FUNCTION_BLOCK FB_RGBLED IMPLEMENTS ITF_SubSystem
VAR_INPUT
	eColor : LEDColor;
END_VAR
VAR
	//Local
	nRedLED : INT;
	nGreenLED : INT;
	nBlueLED : INT;
	
	aErrorTimer : ARRAY [0..5] OF TON;
	
	//ErrorBits
	bRedTemperatureTooHigh : BIT;
	bRedNoSupplyVoltage : BIT;
	bGreenTemperatureTooHigh : BIT;
	bGreenNoSupplyVoltage : BIT;
	bBlueTemperatureTooHigh : BIT;
	bBlueNoSupplyVoltage : BIT;	
END_VAR
VAR CONSTANT
	nMax : INT := 32767;		//Maximum Intensity (100%)
	nMin : INT := 0;			//Off (0%)
END_VAR

CASE eColor OF
	LEDColor.Off:
		nRedLED := nMin;
		nGreenLED := nMin;
		nBlueLED := nMin;
	LEDColor.Red:
		nRedLED := nMax;
		nGreenLED := nMin;
		nBlueLED := nMin;
	LEDColor.Green:
		nRedLED := nMin;
		nGreenLED := nMax;
		nBlueLED := nMin;
	LEDColor.Blue:
		nRedLED := nMin;
		nGreenLED := nMin;
		nBlueLED := nMax;
END_CASE



doSetClampValues();
doGetClampValues();

METHOD PRIVATE doGetClampValues
VAR_INPUT
END_VAR
bRedTemperatureTooHigh := RGBLED.bRedWarning;
bRedNoSupplyVoltage := RGBLED.bRedError;
bGreenTemperatureTooHigh := RGBLED.bGreenWarning;
bGreenNoSupplyVoltage := RGBLED.bGreenError;
bBlueTemperatureTooHigh := RGBLED.bBlueWarning;
bBlueNoSupplyVoltage := RGBLED.bBlueError;
END_METHOD

METHOD PRIVATE doSetClampValues
RGBLED.nRed := nRedLED;
RGBLED.nGreen := nGreenLED;
RGBLED.nBlue := nBlueLED;
END_METHOD

PROPERTY eCondition : SubLevelCondition
GET
IF nErrorID <> 0 THEN
	eCondition := SubLevelCondition.ERROR;
ELSE
	eCondition := SubLevelCondition.RUN;
END_IF
END_GET
END_PROPERTY

PROPERTY nErrorID : UDINT
GET
nErrorID.0 := aErrorTimer[0].Q;
nErrorID.1 := aErrorTimer[1].Q;
nErrorID.2 := aErrorTimer[2].Q;
nErrorID.3 := aErrorTimer[3].Q;
nErrorID.4 := aErrorTimer[4].Q;
nErrorID.5 := aErrorTimer[5].Q;

aErrorTimer[0](IN:=bRedTemperatureTooHigh, PT:=T#5S);
aErrorTimer[1](IN:=bRedNoSupplyVoltage, PT:=T#5S);
aErrorTimer[2](IN:=bGreenTemperatureTooHigh, PT:=T#5S);
aErrorTimer[3](IN:=bGreenNoSupplyVoltage, PT:=T#5S);
aErrorTimer[4](IN:=bBlueTemperatureTooHigh, PT:=T#5S);
aErrorTimer[5](IN:=bBlueNoSupplyVoltage, PT:=T#5S);
END_GET
END_PROPERTY

END_FUNCTION_BLOCK

(* stored: Version 1.1.0.1, ProductVersion 3.1.4024.12
   POU FB_RGBLED: Id {469ae6ce-499d-4fa3-8525-1529c7798012}, SpecialFunc None
   Method doGetClampValues: Id {52eec7f2-2131-4ede-95da-3597bc5e0c67}
   Method doSetClampValues: Id {dbe16808-2cac-4096-8234-89397ca2e1ed}
   Property eCondition: Id {07f8f374-c150-465f-b84c-fb20f0d2bc35}
   Get Get: Id {441c6c85-d8e3-4421-86d4-8b0d5eba7d41}
   Property nErrorID: Id {45849282-d051-426c-bf8e-7a781e21e522}
   Get Get: Id {03514558-8035-44de-ad1f-1de4548a1c2e} *)
